// TIA Portal V20 export
// export: Created 2025-12-01T14:56:13.4875152Z, ExportSetting None, DisplayName Totally Integrated Automation Portal, DisplayVersion V20 Update 3, DisplayName TIA Portal Openness, DisplayVersion V20 Update 3, DisplayName TIA Portal Version Control Interface, DisplayVersion V20 Update 3, DisplayName STEP 7 Professional, DisplayVersion V20 Update 3, DisplayName STEP 7 Safety, DisplayVersion V20 Update 2, DisplayName WinCC Basic/Comfort/Advanced, DisplayVersion V20 Update 3, DisplayName WinCC Professional, DisplayVersion V20 Update 3, DisplayName WinCC Unified, DisplayVersion V20 Update 3
TYPE "UDT_ProtocoloRecMesa"
   STRUCT
      Ord_S00 : Bool;   // Orden de Salida por S0
      Ord_S01 : Bool;   // Orden de Salida por S1
      Ord_S02 : Bool;   // Orden de Salida por S2
      Ord_S03 : Bool;   // Orden de Salida por S3
      Ord_S04 : Bool;   // Orden de Salida por S4
      Ord_Def : Bool;   // Orden por defecto
      Bit_06 : Bool;
      Bit_07 : Bool;
      Bit_10 : Bool;
      Bit_11 : Bool;
      Bit_12 : Bool;
      Bit_13 : Bool;
      Bit_14 : Bool;
      Bit_15 : Bool;
      Bit_16 : Bool;
      EmiOK : Bool;   // Emision OK de la Presencia
   END_STRUCT;
END_TYPE
